TYPE ST_Exhaust :
STRUCT
END_STRUCT
END_TYPE

(* stored: Version 1.1.0.1, ProductVersion 3.1.4024.5
   DUT ST_Exhaust: Id {7837672d-6e2d-420c-b564-587738556bfd} *)
